FUNCTION_BLOCK MachineLogger IMPLEMENTS I_MachineLogger
VAR_INPUT
END_VAR
VAR_OUTPUT
END_VAR
VAR
	fbEventMessage: FB_TcMessage;
	//fbFormatString: FB_FormatString2;
	//sFormat: STRING := 'x = %.2f, z = %.2f';
	
	// Dauer
	tStart: TIME;
END_VAR

METHOD PUBLIC LogBohrung : BOOL
VAR_INPUT
	stPunkt: REFERENCE TO ST_2DPoint;
END_VAR
VAR
	sPara: STRING;
END_VAR
fbEventMessage.CreateEx(TC_EVENTS.BohrEvents.LochGebohrt, 0);
sPara := CONCAT(CONCAT('x = ', LREAL_TO_STRING(stPunkt.x)), CONCAT(', y = ', LREAL_TO_STRING(stPunkt.y)));
fbEventMessage.ipArguments.AddString(sPara);

fbEventMessage.Send(0);
END_METHOD

METHOD PUBLIC LogPunktAngefahren : BOOL
VAR_INPUT
	stPunkt: REFERENCE TO ST_2DPoint;
END_VAR
VAR
	sPara: STRING;
END_VAR
fbEventMessage.CreateEx(TC_EVENTS.BohrEvents.PunktAngefahren, 0);
sPara := CONCAT(CONCAT('x = ', LREAL_TO_STRING(stPunkt.x)), CONCAT(', y = ', LREAL_TO_STRING(stPunkt.y)));
fbEventMessage.ipArguments.AddString(sPara);
fbEventMessage.Send(0);
END_METHOD

METHOD PUBLIC LogStart : BOOL
fbEventMessage.CreateEx(TC_EVENTS.BohrEvents.MaschineGestartet, 0);
fbEventMessage.Send(0);
tStart := TIME();
END_METHOD

METHOD PUBLIC LogStop : BOOL
VAR
	tDauer: TIME;
	sDauer: STRING;
	sPara: STRING;
END_VAR
tDauer := TIME() - tStart;
sDauer := TIME_TO_STRING(tDauer);
fbEventMessage.CreateEx(TC_EVENTS.BohrEvents.MaschineGestoppt, 0);
sPara := CONCAT('Dauer: ', sDauer);
fbEventMessage.ipArguments.AddString(sPara);
fbEventMessage.Send(0);
END_METHOD

END_FUNCTION_BLOCK

(* stored: Version 1.1.0.1, ProductVersion 3.1.4024.3
   POU MachineLogger: Id {b7e329c9-fce1-4e55-b2d7-8b1771ed9387}, SpecialFunc None
   Method LogBohrung: Id {5f642905-dd8a-4b20-9fa4-659bba605ea1}
   Method LogPunktAngefahren: Id {e0c91134-6acc-4108-b4e3-ece266248301}
   Method LogStart: Id {0138aeb6-787b-4d3c-9f8e-6a8a8691ede4}
   Method LogStop: Id {fc3dc073-c4be-48ab-a64b-4dc527bdd047} *)
